% RSLogix 500 project TANKFILL.RSS, saved by version 8.30.00.16 %
PROJECT "UNTITLED"    % processor: Bul.1763 MicroLogix 1100 Series B %

PROGRAM FILES
  LAD 2   3 rungs

DATA FILES
  O0 OUTPUT  4 elements
  I1 INPUT  6 elements
  S2 STATUS  66 elements
  B3 BINARY  1 elements
  T4 TIMER  1 elements
  C5 COUNTER  1 elements
  R6 CONTROL  1 elements
  N7 INTEGER  1 elements
  F8 FLOAT  1 elements

LADDER 2
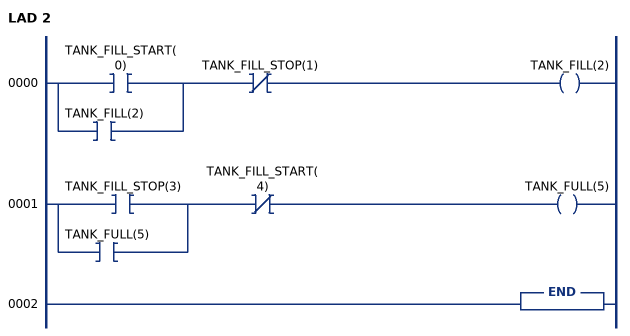
% Rung: 0 %  % edit flag set %
SOR BST XIC TANK_FILL_START(0) NXB XIC TANK_FILL(2) BND XIO TANK_FILL_STOP(1) OTE TANK_FILL(2) EOR
% Rung: 1 %  % edit flag set %
SOR BST XIC TANK_FILL_STOP(3) NXB XIC TANK_FULL(5) BND XIO TANK_FILL_START(4) OTE TANK_FULL(5) EOR
% Rung: 2 %
SOR END EOR

OTHER DOCUMENTED ADDRESSES
  TANK_FULL  
